{attribute 'GeneratedUsingTerminal: EK1200-1388-0000'}
{attribute addProperty VendorId "#x00000002"}
{attribute addProperty BoxType "EK1200-1388-0000"}
{attribute addProperty Description "EK1200-5000 EtherCAT Power supply (2A E-Bus)"}
{attribute addProperty Physics "YK"}
{attribute addProperty Id "EK1200"}
{attribute addProperty CRC "20777801"}
{attribute addProperty Size "0"}
TYPE EK1200_013D0B49 EXTENDS TcoIo.EtcSlaveBoxBase_77A0E4A7 : 
STRUCT
END_STRUCT
END_TYPE

(* stored: Version 1.2.0.0, ProductVersion 3.1.4024.12
   DUT EK1200_013D0B49: Id {80856121-44f9-0aad-2a44-f66c88504450} *)
